ABB RobotStudio station: Solution1_20220203-193357.rsstn

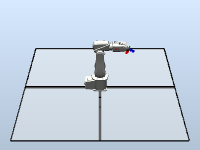
Station Solution1 (saved by RobotStudio 6.8.8307.1040)
Controller IRB_120_3kg_0.58m
  mechanical unit ROB_1: IRB120_3_58__01, 6 joints, base frame (0, 0, 0) mm
Layout (positions relative to the parent item):
  - IRB120_3_58__01 [mechanism, from Robots\IRB120_3_58_G_01.rslib] at (0, 0, 0) mm; joint values [0, 0, 0, 0, 0.5236, 0] (rad or m)
